FUNCTION_BLOCK FB_Stopwatch
VAR_INPUT
END_VAR
VAR_OUTPUT
END_VAR
VAR
	bRunning:		BOOL;
	nIndex:			BYTE;
	tElapsed:		TIME;
END_VAR

IF bRunning THEN
	tElapsed:= tElapsed + M_GetCycletime();
END_IF

METHOD FB_init : BOOL
VAR_INPUT
	bInitRetains : BOOL; // if TRUE, the retain variables are initialized (warm start / cold start)
	bInCopyCode : BOOL;  // if TRUE, the instance afterwards gets moved into the copy code (online change)
END_VAR
VAR
	fbTask:				GETCURTASKINDEX;
END_VAR
fbTask();
nIndex:= fbTask.index;
END_METHOD

METHOD INTERNAL M_GetCycletime : TIME
VAR_INPUT
END_VAR
M_GetCycletime:= LREAL_TO_TIME(UDINT_TO_LREAL(TwinCAT_SystemInfoVarList._TaskInfo[nIndex].CycleTime) / 10000.0);
END_METHOD

METHOD PUBLIC M_Reset : BOOL
VAR_INPUT
END_VAR
bRunning:= FALSE;
tElapsed:= T#0S;
M_Reset:= TRUE;
END_METHOD

METHOD PUBLIC M_Restart : BOOL
VAR_INPUT
END_VAR
bRunning:= TRUE;
tElapsed:= T#0S;
M_Restart:= TRUE;
END_METHOD

METHOD PUBLIC M_Start : BOOL
VAR_INPUT
END_VAR
bRunning:= TRUE;
M_Start:= TRUE;
END_METHOD

METHOD PUBLIC M_Stop : BOOL
VAR_INPUT
END_VAR
bRunning:= FALSE;
M_Stop:= TRUE;
END_METHOD

METHOD PUBLIC M_ToString : String(255)
VAR_INPUT
END_VAR
M_ToString:= TIME_TO_STring(tElapsed);
END_METHOD

PROPERTY PUBLIC P_Elapsed : TIME
GET
P_Elapsed:= tElapsed;
END_GET
END_PROPERTY

PROPERTY PUBLIC P_Running : bool
GET
P_Running:= bRunning;
END_GET
END_PROPERTY

END_FUNCTION_BLOCK

(* stored: Version 1.1.0.1
   POU FB_Stopwatch: Id {ea8d5d03-07a5-0557-320d-b945c7000a26}, SpecialFunc None
   Method FB_init: Id {ab5ba7c6-0946-0698-3d6e-a909fd4dfd48}
   Method M_GetCycletime: Id {338c9ee5-70a2-0048-11a8-0849581c2877}
   Method M_Reset: Id {ba944a76-c6c6-09c2-3ee3-b7bdd8ffc878}
   Method M_Restart: Id {c046b838-c816-017e-2d5a-07c04968c6b0}
   Method M_Start: Id {c4894435-be15-0c3e-1ce6-e45af90b931c}
   Method M_Stop: Id {ad8d41dc-63d6-002e-19b5-772bdd2bad6b}
   Method M_ToString: Id {a5c47b34-177a-0110-3c5e-fa58afcd8a30}
   Property P_Elapsed: Id {2ad96b99-8cf7-00e2-36db-08df0650367e}
   Get Get: Id {97a5abbf-958d-0c6a-3e54-414d0b1ac9db}
   Property P_Running: Id {02d97fa5-9906-063b-0201-0418a51019c9}
   Get Get: Id {e2e5c92d-51c7-0242-128c-d32a8f0e272e} *)
